(* PLC project SafeLOGIC, BrAutomation SafeDESIGNER  5.24.1.0 *)
(* stored: companyURL http://www.br-automation.com, creationDateTime Fri Nov 28 14:16:19 2025 *)

PROGRAM KeepAMM_2s

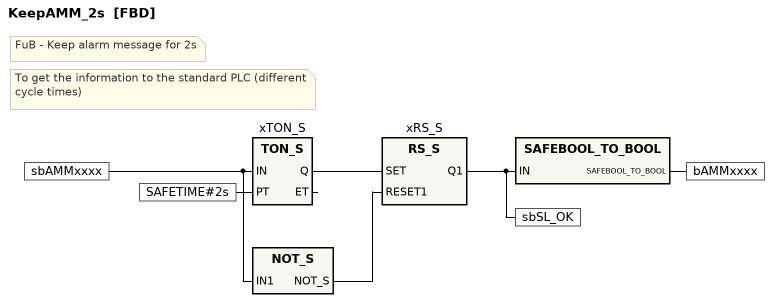
(* FBD diagram, written out as Structured Text *)
(* FuB - Keep alarm message for 2s *)
(* To get the information to the standard PLC (different cycle times) *)
xTON_S(IN := sbAMMxxxx, PT := SAFETIME#2s);
xRS_S(SET := xTON_S.Q, RESET1 := NOT_S(sbAMMxxxx));
bAMMxxxx := SAFEBOOL_TO_BOOL(xRS_S.Q1);
sbSL_OK := xRS_S.Q1;
END_PROGRAM
